FUNCTION_BLOCK FB_FaultChecker
VAR_INPUT
END_VAR
VAR_OUTPUT
END_VAR
VAR_IN_OUT
    aFaultsToCheck  : ARRAY [*] OF FB_FaultEvent;
END_VAR
VAR CONSTANT
	//Constants as defined in Pulse Pisa Manuals
    //MAX_FAULTS : USINT            := 255;     
END_VAR

VAR
	nIdx   : DINT;
    nSum   : DINT;
	nLastWrittenIndex :UINT:=0;
	
	
	//aFaultsToCheck : ARRAY[1..MAX_NUMBER_OF_CHANNELS] OF CircuitBreakerStatus := [MAX_NUMBER_OF_CHANNELS(CircuitBreakerStatus.UNKNOWN)]; 
END_VAR

FOR nIdx := LOWER_BOUND(aFaultsToCheck,1) TO UPPER_BOUND(aFaultsToCheck,1) DO
    aFaultsToCheck[nIdx].Update();
END_FOR;

METHOD PUBLIC AddEvent
VAR_INPUT
	fbEvent : Pointer TO FB_FaultEvent;
END_VAR
aFaultsToCheck[nLastWrittenIndex]:=fbEvent^;
nLastWrittenIndex := nLastWrittenIndex +1;
END_METHOD

METHOD GetActiveEventCount : UINT
VAR
	nActiveEventCount:UINT:=0;
END_VAR
FOR nIdx := LOWER_BOUND(aFaultsToCheck,1) TO UPPER_BOUND(aFaultsToCheck,1) DO
	IF(    aFaultsToCheck[nIdx].Active())THEN
		nActiveEventCount:=nActiveEventCount+1;
	END_IF
END_FOR;
GetActiveEventCount:=nActiveEventCount;
END_METHOD

METHOD PUBLIC GetFirstActiveEvent : REFERENCE TO FB_FaultEvent
VAR_INPUT
END_VAR
FOR nIdx := LOWER_BOUND(aFaultsToCheck,1) TO UPPER_BOUND(aFaultsToCheck,1) DO
	IF(aFaultsToCheck[nIdx].Active()) THEN
		GetFirstActiveEvent:=aFaultsToCheck[nIdx];
		EXIT;
	END_IF
END_FOR;
END_METHOD

END_FUNCTION_BLOCK

(* stored: Version 1.1.0.1, ProductVersion 3.1.4024.15
   POU FB_FaultChecker: Id {81627131-cc2a-4f8a-9243-c943820076da}, SpecialFunc None
   Method AddEvent: Id {d7e83bef-d5e1-4fe8-b79a-89c8086b3844}
   Method GetActiveEventCount: Id {cd32fd0b-e511-4ff1-8c9d-ef12759e2e01}
   Method GetFirstActiveEvent: Id {a193127a-8663-4ec2-a895-c7ca5ea2f347} *)
